TYPE PiperModuleInternal :
STRUCT
	machine : REFERENCE TO Piper;
	context : IPluginRunner;
	registered : BOOL;
	response : RESPONSE_STATE;
	requestSubstate : ULINT;
	previousSubstate : ULINT;
	previousSubstateAsync : ULINT;
	skipsSync : PiperImplements;
	skipsAsync : PiperImplements;	
	requestNumber : DINT;
END_STRUCT
END_TYPE

(* stored: Version 1.1.0.1
   DUT PiperModuleInternal: Id {d334c6b3-1691-0666-3b67-eb120f59ab5a} *)
